TYPE ST_LED :
STRUCT
	eLEDState: E_LED_STATE;
	eLEDErrorStatus: E_LED_Errors;
	bRequestApproved: BOOL;
	fbTimer: TON := (IN:=FALSE);
	fbTrigger: R_TRIG := (CLK:=fbTimer.Q);
	tTarget: TIME;
	color: STRING;
END_STRUCT
END_TYPE

(* stored: Version 1.1.0.1, ProductVersion 3.1.4022.12
   DUT ST_LED: Id {1a645526-e5f7-497b-ad08-d5a697b15633} *)
